{attribute 'GeneratedUsingTerminal: EP2339-0003-0016'}
{attribute addProperty BoxType "EP2339-0003-0016"}
{attribute addProperty Description "EP2339-0003 16 Ch. Dig. Input/Output 24V, 0,5A, 10-Pole Plug Connector"}
{attribute addProperty Physics "YY"}
{attribute addProperty Id "DI_Inputs_Channel_1AT %I*DI_Inputs_Channel_91AC31B711DI_Inputs_Channel_2AT %I*DI_Inputs_Channel_91AC31B711DO_Outputs_Channel_1AT %Q*DO_Outputs_Channel_28AC1A9E8DO_Outputs_Channel_2AT %Q*DO_Outputs_Channel_28AC1A9E8WcStateAT %I*WcState_9091E0EB2InfoDataAT %I*InfoData_32EB74EA10"}
{attribute addProperty CRC "2998276840"}
{attribute addProperty Size "50"}
TYPE EP2339_B2B612E8 EXTENDS EtcSlaveBoxBase_77A0E4A7 :
STRUCT
	{attribute addProperty Name "DI_Inputs_Channel_1"}
	DI_Inputs_Channel_1 : DI_Inputs_Channel_91AC31B7;
	{attribute addProperty Name "DI_Inputs_Channel_2"}
	DI_Inputs_Channel_2 : DI_Inputs_Channel_91AC31B7;
	{attribute addProperty Name "DO_Outputs_Channel_1"}
	DO_Outputs_Channel_1 : DO_Outputs_Channel_28AC1A9E;
	{attribute addProperty Name "DO_Outputs_Channel_2"}
	DO_Outputs_Channel_2 : DO_Outputs_Channel_28AC1A9E;
	{attribute addProperty Name "WcState"}
	WcState : WcState_9091E0EB;
	{attribute addProperty Name "InfoData"}
	InfoData : InfoData_32EB74EA;
END_STRUCT
END_TYPE

(* stored: Version 1.2.0.0, ProductVersion 3.1.4024.11
   DUT EP2339_B2B612E8: Id {6ecd9473-7088-4c0e-b939-4e81a10432f8} *)
